{attribute 'qualified_only'}
VAR_GLOBAL INTERNAL
	{attribute 'ExpandFully'} 
	entry				: ARRAY[1..Param.RECEIVER_CAP] OF _BroadcastStruct;
	iSignal				: ARRAY[1..Param.SIGNAL_CAP] OF I_SignalNode;
	iFirst				: I_SignalNode;
	nRecLen				: UDINT;
	nSignalLen			: UDINT;
	bRegLock			: BOOL;
END_VAR

(* stored: Version 1.1.0.1
   GVL _Broadcast: Id {c6aa29cd-8dd8-49f5-821b-ac6fe8fd276f} *)
